PROGRAM MAIN
VAR
END_VAR

END_PROGRAM

(* stored: Version 1.1.0.1
   POU MAIN: Id {e5e08434-e2a7-4277-93b2-315b6105b566} *)
